ABB RAPID module: Module1.mod

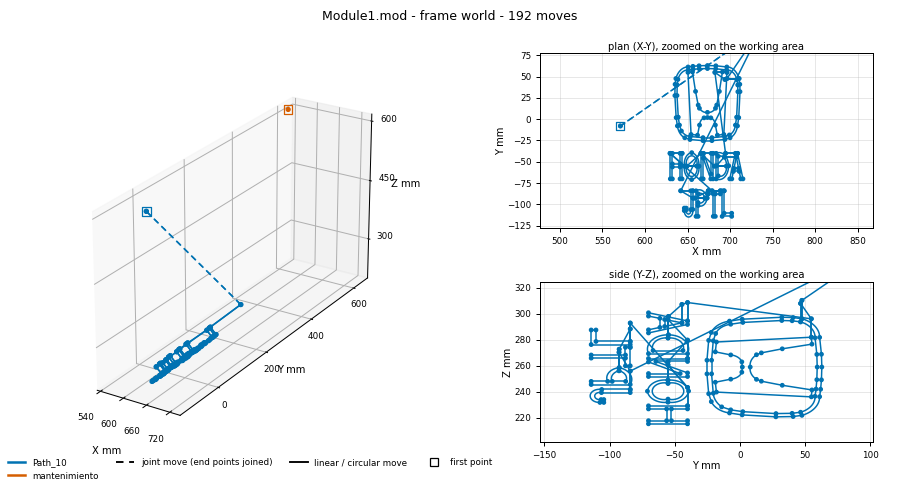
[picture p0: tool path of Module1.mod in frame world, 192 of 192 moves have a stored position in this frame; points joined in program order, loops and branches not executed]
MODULE Module1
        CONST robtarget Target_10:=[[0,0,-20],[0.707106781,0,0,0.707106781],[0,0,0,0],[9E+09,9E+09,9E+09,9E+09,9E+09,9E+09]];
    CONST robtarget Target_20:=[[59.453,57.54,-20],[0.707106781,0,0,0.707106781],[0,0,0,0],[9E+09,9E+09,9E+09,9E+09,9E+09,9E+09]];
    CONST robtarget Target_30:=[[59.453,57.54,0],[0.707106781,0,0,0.707106781],[0,0,0,0],[9E+09,9E+09,9E+09,9E+09,9E+09,9E+09]];
    CONST robtarget Target_40:=[[66.223,56.236,0],[0.707106781,0,0,0.707106781],[0,0,0,0],[9E+09,9E+09,9E+09,9E+09,9E+09,9E+09]];
    CONST robtarget Target_50:=[[74.887,55.915,0],[0.707106781,0,0,0.707106781],[0,0,0,0],[9E+09,9E+09,9E+09,9E+09,9E+09,9E+09]];
    CONST robtarget Target_60:=[[105.351,58.027,0],[0.707106781,0,0,0.707106781],[0,0,0,0],[9E+09,9E+09,9E+09,9E+09,9E+09,9E+09]];
    CONST robtarget Target_70:=[[115.083,60.098,0],[0.707106781,0,0,0.707106781],[0,0,0,0],[9E+09,9E+09,9E+09,9E+09,9E+09,9E+09]];
    CONST robtarget Target_90:=[[123.324,63.988,0],[0.707106781,0,0,0.707106781],[0,0,0,0],[9E+09,9E+09,9E+09,9E+09,9E+09,9E+09]];
    CONST robtarget Target_100:=[[129.054,72.401,0],[0.707106781,0,0,0.707106781],[0,0,0,0],[9E+09,9E+09,9E+09,9E+09,9E+09,9E+09]];
    CONST robtarget Target_110:=[[131.081,81.035,0],[0.707106781,0,0,0.707106781],[0,0,0,0],[9E+09,9E+09,9E+09,9E+09,9E+09,9E+09]];
    CONST robtarget Target_120:=[[132.397,102.578,0],[0.707106781,0,0,0.707106781],[0,0,0,0],[9E+09,9E+09,9E+09,9E+09,9E+09,9E+09]];
    CONST robtarget Target_130:=[[132.397,117.423,0],[0.707106781,0,0,0.707106781],[0,0,0,0],[9E+09,9E+09,9E+09,9E+09,9E+09,9E+09]];
    CONST robtarget Target_140:=[[131.081,138.966,0],[0.707106781,0,0,0.707106781],[0,0,0,0],[9E+09,9E+09,9E+09,9E+09,9E+09,9E+09]];
    CONST robtarget Target_150:=[[129.054,147.6,0],[0.707106781,0,0,0.707106781],[0,0,0,0],[9E+09,9E+09,9E+09,9E+09,9E+09,9E+09]];
    CONST robtarget Target_160:=[[123.324,156.012,0],[0.707106781,0,0,0.707106781],[0,0,0,0],[9E+09,9E+09,9E+09,9E+09,9E+09,9E+09]];
    CONST robtarget Target_170:=[[115.083,159.903,0],[0.707106781,0,0,0.707106781],[0,0,0,0],[9E+09,9E+09,9E+09,9E+09,9E+09,9E+09]];
    CONST robtarget Target_180:=[[105.351,161.974,0],[0.707106781,0,0,0.707106781],[0,0,0,0],[9E+09,9E+09,9E+09,9E+09,9E+09,9E+09]];
    CONST robtarget Target_190:=[[79.466,164.086,0],[0.707106781,0,0,0.707106781],[0,0,0,0],[9E+09,9E+09,9E+09,9E+09,9E+09,9E+09]];
    CONST robtarget Target_200:=[[66.223,163.764,0],[0.707106781,0,0,0.707106781],[0,0,0,0],[9E+09,9E+09,9E+09,9E+09,9E+09,9E+09]];
    CONST robtarget Target_210:=[[59.453,162.461,0],[0.707106781,0,0,0.707106781],[0,0,0,0],[9E+09,9E+09,9E+09,9E+09,9E+09,9E+09]];
    CONST robtarget Target_220:=[[48.886,153.475,0],[0.707106781,0,0,0.707106781],[0,0,0,0],[9E+09,9E+09,9E+09,9E+09,9E+09,9E+09]];
    CONST robtarget Target_230:=[[45.864,142.196,0],[0.707106781,0,0,0.707106781],[0,0,0,0],[9E+09,9E+09,9E+09,9E+09,9E+09,9E+09]];
    CONST robtarget Target_240:=[[45.105,134.144,0],[0.707106781,0,0,0.707106781],[0,0,0,0],[9E+09,9E+09,9E+09,9E+09,9E+09,9E+09]];
    CONST robtarget Target_250:=[[44.474,123.905,0],[0.707106781,0,0,0.707106781],[0,0,0,0],[9E+09,9E+09,9E+09,9E+09,9E+09,9E+09]];
    CONST robtarget Target_260:=[[44.178,110,0],[0.707106781,0,0,0.707106781],[0,0,0,0],[9E+09,9E+09,9E+09,9E+09,9E+09,9E+09]];
    CONST robtarget Target_270:=[[44.474,96.095,0],[0.707106781,0,0,0.707106781],[0,0,0,0],[9E+09,9E+09,9E+09,9E+09,9E+09,9E+09]];
    CONST robtarget Target_280:=[[45.864,77.804,0],[0.707106781,0,0,0.707106781],[0,0,0,0],[9E+09,9E+09,9E+09,9E+09,9E+09,9E+09]];
    CONST robtarget Target_290:=[[48.886,66.526,0],[0.707106781,0,0,0.707106781],[0,0,0,0],[9E+09,9E+09,9E+09,9E+09,9E+09,9E+09]];
    CONST robtarget Target_300:=[[59.453,57.54,0],[0.707106781,0,0,0.707106781],[0,0,0,0],[9E+09,9E+09,9E+09,9E+09,9E+09,9E+09]];
    CONST robtarget Target_310:=[[59.453,57.54,-20],[0.707106781,0,0,0.707106781],[0,0,0,0],[9E+09,9E+09,9E+09,9E+09,9E+09,9E+09]];
    CONST robtarget Target_320:=[[60.499,60.925,-20],[0.707106781,0,0,0.707106781],[0,0,0,0],[9E+09,9E+09,9E+09,9E+09,9E+09,9E+09]];
    CONST robtarget Target_330:=[[60.499,60.925,0],[0.707106781,0,0,0.707106781],[0,0,0,0],[9E+09,9E+09,9E+09,9E+09,9E+09,9E+09]];
    CONST robtarget Target_340:=[[67.002,59.732,0],[0.707106781,0,0,0.707106781],[0,0,0,0],[9E+09,9E+09,9E+09,9E+09,9E+09,9E+09]];
    CONST robtarget Target_350:=[[74.944,59.458,0],[0.707106781,0,0,0.707106781],[0,0,0,0],[9E+09,9E+09,9E+09,9E+09,9E+09,9E+09]];
    CONST robtarget Target_360:=[[104.86,61.536,0],[0.707106781,0,0,0.707106781],[0,0,0,0],[9E+09,9E+09,9E+09,9E+09,9E+09,9E+09]];
    CONST robtarget Target_370:=[[114.154,63.519,0],[0.707106781,0,0,0.707106781],[0,0,0,0],[9E+09,9E+09,9E+09,9E+09,9E+09,9E+09]];
    CONST robtarget Target_380:=[[121.091,66.742,0],[0.707106781,0,0,0.707106781],[0,0,0,0],[9E+09,9E+09,9E+09,9E+09,9E+09,9E+09]];
    CONST robtarget Target_390:=[[125.713,73.58,0],[0.707106781,0,0,0.707106781],[0,0,0,0],[9E+09,9E+09,9E+09,9E+09,9E+09,9E+09]];
    CONST robtarget Target_400:=[[127.565,81.47,0],[0.707106781,0,0,0.707106781],[0,0,0,0],[9E+09,9E+09,9E+09,9E+09,9E+09,9E+09]];
    CONST robtarget Target_410:=[[128.854,102.618,0],[0.707106781,0,0,0.707106781],[0,0,0,0],[9E+09,9E+09,9E+09,9E+09,9E+09,9E+09]];
    CONST robtarget Target_420:=[[128.854,117.382,0],[0.707106781,0,0,0.707106781],[0,0,0,0],[9E+09,9E+09,9E+09,9E+09,9E+09,9E+09]];
    CONST robtarget Target_430:=[[127.565,138.53,0],[0.707106781,0,0,0.707106781],[0,0,0,0],[9E+09,9E+09,9E+09,9E+09,9E+09,9E+09]];
    CONST robtarget Target_440:=[[125.713,146.42,0],[0.707106781,0,0,0.707106781],[0,0,0,0],[9E+09,9E+09,9E+09,9E+09,9E+09,9E+09]];
    CONST robtarget Target_450:=[[121.091,153.258,0],[0.707106781,0,0,0.707106781],[0,0,0,0],[9E+09,9E+09,9E+09,9E+09,9E+09,9E+09]];
    CONST robtarget Target_460:=[[114.154,156.482,0],[0.707106781,0,0,0.707106781],[0,0,0,0],[9E+09,9E+09,9E+09,9E+09,9E+09,9E+09]];
    CONST robtarget Target_470:=[[104.86,158.465,0],[0.707106781,0,0,0.707106781],[0,0,0,0],[9E+09,9E+09,9E+09,9E+09,9E+09,9E+09]];
    CONST robtarget Target_480:=[[79.395,160.544,0],[0.707106781,0,0,0.707106781],[0,0,0,0],[9E+09,9E+09,9E+09,9E+09,9E+09,9E+09]];
    CONST robtarget Target_490:=[[67.002,160.268,0],[0.707106781,0,0,0.707106781],[0,0,0,0],[9E+09,9E+09,9E+09,9E+09,9E+09,9E+09]];
    CONST robtarget Target_500:=[[60.499,159.075,0],[0.707106781,0,0,0.707106781],[0,0,0,0],[9E+09,9E+09,9E+09,9E+09,9E+09,9E+09]];
    CONST robtarget Target_510:=[[52.059,151.898,0],[0.707106781,0,0,0.707106781],[0,0,0,0],[9E+09,9E+09,9E+09,9E+09,9E+09,9E+09]];
    CONST robtarget Target_520:=[[49.379,141.75,0],[0.707106781,0,0,0.707106781],[0,0,0,0],[9E+09,9E+09,9E+09,9E+09,9E+09,9E+09]];
    CONST robtarget Target_530:=[[48.642,133.935,0],[0.707106781,0,0,0.707106781],[0,0,0,0],[9E+09,9E+09,9E+09,9E+09,9E+09,9E+09]];
    CONST robtarget Target_540:=[[48.013,123.721,0],[0.707106781,0,0,0.707106781],[0,0,0,0],[9E+09,9E+09,9E+09,9E+09,9E+09,9E+09]];
    CONST robtarget Target_550:=[[47.721,110,0],[0.707106781,0,0,0.707106781],[0,0,0,0],[9E+09,9E+09,9E+09,9E+09,9E+09,9E+09]];
    CONST robtarget Target_560:=[[48.013,96.28,0],[0.707106781,0,0,0.707106781],[0,0,0,0],[9E+09,9E+09,9E+09,9E+09,9E+09,9E+09]];
    CONST robtarget Target_570:=[[49.379,78.251,0],[0.707106781,0,0,0.707106781],[0,0,0,0],[9E+09,9E+09,9E+09,9E+09,9E+09,9E+09]];
    CONST robtarget Target_580:=[[52.059,68.102,0],[0.707106781,0,0,0.707106781],[0,0,0,0],[9E+09,9E+09,9E+09,9E+09,9E+09,9E+09]];
    CONST robtarget Target_590:=[[60.499,60.925,0],[0.707106781,0,0,0.707106781],[0,0,0,0],[9E+09,9E+09,9E+09,9E+09,9E+09,9E+09]];
    CONST robtarget Target_600:=[[60.499,60.925,-20],[0.707106781,0,0,0.707106781],[0,0,0,0],[9E+09,9E+09,9E+09,9E+09,9E+09,9E+09]];
    CONST robtarget Target_610:=[[52.233,77.609,-20],[0.707106781,0,0,0.707106781],[0,0,0,0],[9E+09,9E+09,9E+09,9E+09,9E+09,9E+09]];
    CONST robtarget Target_620:=[[52.233,77.609,0],[0.707106781,0,0,0.707106781],[0,0,0,0],[9E+09,9E+09,9E+09,9E+09,9E+09,9E+09]];
    CONST robtarget Target_630:=[[125.12,82.794,0],[0.707106781,0,0,0.707106781],[0,0,0,0],[9E+09,9E+09,9E+09,9E+09,9E+09,9E+09]];
    CONST robtarget Target_640:=[[125.974,93.513,0],[0.707106781,0,0,0.707106781],[0,0,0,0],[9E+09,9E+09,9E+09,9E+09,9E+09,9E+09]];
    CONST robtarget Target_650:=[[114.117,96.833,0],[0.707106781,0,0,0.707106781],[0,0,0,0],[9E+09,9E+09,9E+09,9E+09,9E+09,9E+09]];
    CONST robtarget Target_660:=[[109.268,98.854,0],[0.707106781,0,0,0.707106781],[0,0,0,0],[9E+09,9E+09,9E+09,9E+09,9E+09,9E+09]];
    CONST robtarget Target_670:=[[105.623,104.378,0],[0.707106781,0,0,0.707106781],[0,0,0,0],[9E+09,9E+09,9E+09,9E+09,9E+09,9E+09]];
    CONST robtarget Target_680:=[[105.23,110,0],[0.707106781,0,0,0.707106781],[0,0,0,0],[9E+09,9E+09,9E+09,9E+09,9E+09,9E+09]];
    CONST robtarget Target_690:=[[105.623,115.622,0],[0.707106781,0,0,0.707106781],[0,0,0,0],[9E+09,9E+09,9E+09,9E+09,9E+09,9E+09]];
    CONST robtarget Target_700:=[[109.268,121.147,0],[0.707106781,0,0,0.707106781],[0,0,0,0],[9E+09,9E+09,9E+09,9E+09,9E+09,9E+09]];
    CONST robtarget Target_710:=[[114.117,123.168,0],[0.707106781,0,0,0.707106781],[0,0,0,0],[9E+09,9E+09,9E+09,9E+09,9E+09,9E+09]];
    CONST robtarget Target_720:=[[125.974,126.488,0],[0.707106781,0,0,0.707106781],[0,0,0,0],[9E+09,9E+09,9E+09,9E+09,9E+09,9E+09]];
    CONST robtarget Target_730:=[[125.12,137.207,0],[0.707106781,0,0,0.707106781],[0,0,0,0],[9E+09,9E+09,9E+09,9E+09,9E+09,9E+09]];
    CONST robtarget Target_740:=[[52.233,142.391,0],[0.707106781,0,0,0.707106781],[0,0,0,0],[9E+09,9E+09,9E+09,9E+09,9E+09,9E+09]];
    CONST robtarget Target_750:=[[51.773,134.866,0],[0.707106781,0,0,0.707106781],[0,0,0,0],[9E+09,9E+09,9E+09,9E+09,9E+09,9E+09]];
    CONST robtarget Target_760:=[[74.57,129.805,0],[0.707106781,0,0,0.707106781],[0,0,0,0],[9E+09,9E+09,9E+09,9E+09,9E+09,9E+09]];
    CONST robtarget Target_770:=[[90.628,125.39,0],[0.707106781,0,0,0.707106781],[0,0,0,0],[9E+09,9E+09,9E+09,9E+09,9E+09,9E+09]];
    CONST robtarget Target_780:=[[94.375,123.358,0],[0.707106781,0,0,0.707106781],[0,0,0,0],[9E+09,9E+09,9E+09,9E+09,9E+09,9E+09]];
    CONST robtarget Target_790:=[[98.757,116.086,0],[0.707106781,0,0,0.707106781],[0,0,0,0],[9E+09,9E+09,9E+09,9E+09,9E+09,9E+09]];
    CONST robtarget Target_800:=[[99.17,110,0],[0.707106781,0,0,0.707106781],[0,0,0,0],[9E+09,9E+09,9E+09,9E+09,9E+09,9E+09]];
    CONST robtarget Target_810:=[[98.757,103.915,0],[0.707106781,0,0,0.707106781],[0,0,0,0],[9E+09,9E+09,9E+09,9E+09,9E+09,9E+09]];
    CONST robtarget Target_820:=[[94.375,96.643,0],[0.707106781,0,0,0.707106781],[0,0,0,0],[9E+09,9E+09,9E+09,9E+09,9E+09,9E+09]];
    CONST robtarget Target_830:=[[90.628,94.611,0],[0.707106781,0,0,0.707106781],[0,0,0,0],[9E+09,9E+09,9E+09,9E+09,9E+09,9E+09]];
    CONST robtarget Target_840:=[[74.57,90.195,0],[0.707106781,0,0,0.707106781],[0,0,0,0],[9E+09,9E+09,9E+09,9E+09,9E+09,9E+09]];
    CONST robtarget Target_850:=[[51.773,85.135,0],[0.707106781,0,0,0.707106781],[0,0,0,0],[9E+09,9E+09,9E+09,9E+09,9E+09,9E+09]];
    CONST robtarget Target_860:=[[52.233,77.609,0],[0.707106781,0,0,0.707106781],[0,0,0,0],[9E+09,9E+09,9E+09,9E+09,9E+09,9E+09]];
    CONST robtarget Target_870:=[[52.233,77.609,-20],[0.707106781,0,0,0.707106781],[0,0,0,0],[9E+09,9E+09,9E+09,9E+09,9E+09,9E+09]];
    CONST robtarget Target_880:=[[147.311,59.932,-20],[0.707106781,0,0,0.707106781],[0,0,0,0],[9E+09,9E+09,9E+09,9E+09,9E+09,9E+09]];
    CONST robtarget Target_890:=[[147.311,59.932,0],[0.707106781,0,0,0.707106781],[0,0,0,0],[9E+09,9E+09,9E+09,9E+09,9E+09,9E+09]];
    CONST robtarget Target_900:=[[177.311,51.036,0],[0.707106781,0,0,0.707106781],[0,0,0,0],[9E+09,9E+09,9E+09,9E+09,9E+09,9E+09]];
    CONST robtarget Target_910:=[[177.311,54.661,0],[0.707106781,0,0,0.707106781],[0,0,0,0],[9E+09,9E+09,9E+09,9E+09,9E+09,9E+09]];
    CONST robtarget Target_920:=[[168.583,57.094,0],[0.707106781,0,0,0.707106781],[0,0,0,0],[9E+09,9E+09,9E+09,9E+09,9E+09,9E+09]];
    CONST robtarget Target_930:=[[168.583,66.943,0],[0.707106781,0,0,0.707106781],[0,0,0,0],[9E+09,9E+09,9E+09,9E+09,9E+09,9E+09]];
    CONST robtarget Target_940:=[[177.311,69.542,0],[0.707106781,0,0,0.707106781],[0,0,0,0],[9E+09,9E+09,9E+09,9E+09,9E+09,9E+09]];
    CONST robtarget Target_950:=[[177.311,72.976,0],[0.707106781,0,0,0.707106781],[0,0,0,0],[9E+09,9E+09,9E+09,9E+09,9E+09,9E+09]];
    CONST robtarget Target_960:=[[147.311,63.747,0],[0.707106781,0,0,0.707106781],[0,0,0,0],[9E+09,9E+09,9E+09,9E+09,9E+09,9E+09]];
    CONST robtarget Target_970:=[[147.311,59.932,0],[0.707106781,0,0,0.707106781],[0,0,0,0],[9E+09,9E+09,9E+09,9E+09,9E+09,9E+09]];
    CONST robtarget Target_980:=[[147.311,59.932,-20],[0.707106781,0,0,0.707106781],[0,0,0,0],[9E+09,9E+09,9E+09,9E+09,9E+09,9E+09]];
    CONST robtarget Target_990:=[[151.627,61.982,-20],[0.707106781,0,0,0.707106781],[0,0,0,0],[9E+09,9E+09,9E+09,9E+09,9E+09,9E+09]];
    CONST robtarget Target_1000:=[[151.627,61.982,0],[0.707106781,0,0,0.707106781],[0,0,0,0],[9E+09,9E+09,9E+09,9E+09,9E+09,9E+09]];
    CONST robtarget Target_1010:=[[164.91,65.941,0],[0.707106781,0,0,0.707106781],[0,0,0,0],[9E+09,9E+09,9E+09,9E+09,9E+09,9E+09]];
    CONST robtarget Target_1020:=[[164.91,58.31,0],[0.707106781,0,0,0.707106781],[0,0,0,0],[9E+09,9E+09,9E+09,9E+09,9E+09,9E+09]];
    CONST robtarget Target_1030:=[[151.627,61.982,0],[0.707106781,0,0,0.707106781],[0,0,0,0],[9E+09,9E+09,9E+09,9E+09,9E+09,9E+09]];
    CONST robtarget Target_1040:=[[151.627,61.982,-20],[0.707106781,0,0,0.707106781],[0,0,0,0],[9E+09,9E+09,9E+09,9E+09,9E+09,9E+09]];
    CONST robtarget Target_1050:=[[161.977,75.051,-20],[0.707106781,0,0,0.707106781],[0,0,0,0],[9E+09,9E+09,9E+09,9E+09,9E+09,9E+09]];
    CONST robtarget Target_1060:=[[161.977,75.051,0],[0.707106781,0,0,0.707106781],[0,0,0,0],[9E+09,9E+09,9E+09,9E+09,9E+09,9E+09]];
    CONST robtarget Target_1070:=[[177.311,85.567,0],[0.707106781,0,0,0.707106781],[0,0,0,0],[9E+09,9E+09,9E+09,9E+09,9E+09,9E+09]];
    CONST robtarget Target_1080:=[[177.311,95.44,0],[0.707106781,0,0,0.707106781],[0,0,0,0],[9E+09,9E+09,9E+09,9E+09,9E+09,9E+09]];
    CONST robtarget Target_1090:=[[147.311,95.44,0],[0.707106781,0,0,0.707106781],[0,0,0,0],[9E+09,9E+09,9E+09,9E+09,9E+09,9E+09]];
    CONST robtarget Target_1100:=[[147.311,85.424,0],[0.707106781,0,0,0.707106781],[0,0,0,0],[9E+09,9E+09,9E+09,9E+09,9E+09,9E+09]];
    CONST robtarget Target_1110:=[[161.977,75.051,0],[0.707106781,0,0,0.707106781],[0,0,0,0],[9E+09,9E+09,9E+09,9E+09,9E+09,9E+09]];
    CONST robtarget Target_1120:=[[161.977,75.051,-20],[0.707106781,0,0,0.707106781],[0,0,0,0],[9E+09,9E+09,9E+09,9E+09,9E+09,9E+09]];
    CONST robtarget Target_1130:=[[162.311,78.437,-20],[0.707106781,0,0,0.707106781],[0,0,0,0],[9E+09,9E+09,9E+09,9E+09,9E+09,9E+09]];
    CONST robtarget Target_1140:=[[162.311,78.437,0],[0.707106781,0,0,0.707106781],[0,0,0,0],[9E+09,9E+09,9E+09,9E+09,9E+09,9E+09]];
    CONST robtarget Target_1150:=[[173.806,85.591,0],[0.707106781,0,0,0.707106781],[0,0,0,0],[9E+09,9E+09,9E+09,9E+09,9E+09,9E+09]];
    CONST robtarget Target_1160:=[[173.806,92.054,0],[0.707106781,0,0,0.707106781],[0,0,0,0],[9E+09,9E+09,9E+09,9E+09,9E+09,9E+09]];
    CONST robtarget Target_1170:=[[150.817,92.054,0],[0.707106781,0,0,0.707106781],[0,0,0,0],[9E+09,9E+09,9E+09,9E+09,9E+09,9E+09]];
    CONST robtarget Target_1180:=[[150.817,85.806,0],[0.707106781,0,0,0.707106781],[0,0,0,0],[9E+09,9E+09,9E+09,9E+09,9E+09,9E+09]];
    CONST robtarget Target_1190:=[[162.311,78.437,0],[0.707106781,0,0,0.707106781],[0,0,0,0],[9E+09,9E+09,9E+09,9E+09,9E+09,9E+09]];
    CONST robtarget Target_1200:=[[162.311,78.437,-20],[0.707106781,0,0,0.707106781],[0,0,0,0],[9E+09,9E+09,9E+09,9E+09,9E+09,9E+09]];
    CONST robtarget Target_1210:=[[147.311,100.734,-20],[0.707106781,0,0,0.707106781],[0,0,0,0],[9E+09,9E+09,9E+09,9E+09,9E+09,9E+09]];
    CONST robtarget Target_1220:=[[147.311,100.734,0],[0.707106781,0,0,0.707106781],[0,0,0,0],[9E+09,9E+09,9E+09,9E+09,9E+09,9E+09]];
    CONST robtarget Target_1230:=[[177.311,100.734,0],[0.707106781,0,0,0.707106781],[0,0,0,0],[9E+09,9E+09,9E+09,9E+09,9E+09,9E+09]];
    CONST robtarget Target_1240:=[[177.311,104.455,0],[0.707106781,0,0,0.707106781],[0,0,0,0],[9E+09,9E+09,9E+09,9E+09,9E+09,9E+09]];
    CONST robtarget Target_1250:=[[152.963,117.07,0],[0.707106781,0,0,0.707106781],[0,0,0,0],[9E+09,9E+09,9E+09,9E+09,9E+09,9E+09]];
    CONST robtarget Target_1260:=[[177.311,117.07,0],[0.707106781,0,0,0.707106781],[0,0,0,0],[9E+09,9E+09,9E+09,9E+09,9E+09,9E+09]];
    CONST robtarget Target_1270:=[[177.311,120.289,0],[0.707106781,0,0,0.707106781],[0,0,0,0],[9E+09,9E+09,9E+09,9E+09,9E+09,9E+09]];
    CONST robtarget Target_1280:=[[147.311,120.289,0],[0.707106781,0,0,0.707106781],[0,0,0,0],[9E+09,9E+09,9E+09,9E+09,9E+09,9E+09]];
    CONST robtarget Target_1290:=[[147.311,116.354,0],[0.707106781,0,0,0.707106781],[0,0,0,0],[9E+09,9E+09,9E+09,9E+09,9E+09,9E+09]];
    CONST robtarget Target_1300:=[[171.659,103.954,0],[0.707106781,0,0,0.707106781],[0,0,0,0],[9E+09,9E+09,9E+09,9E+09,9E+09,9E+09]];
    CONST robtarget Target_1310:=[[147.311,103.954,0],[0.707106781,0,0,0.707106781],[0,0,0,0],[9E+09,9E+09,9E+09,9E+09,9E+09,9E+09]];
    CONST robtarget Target_1320:=[[147.311,100.734,0],[0.707106781,0,0,0.707106781],[0,0,0,0],[9E+09,9E+09,9E+09,9E+09,9E+09,9E+09]];
    CONST robtarget Target_1330:=[[147.311,100.734,-20],[0.707106781,0,0,0.707106781],[0,0,0,0],[9E+09,9E+09,9E+09,9E+09,9E+09,9E+09]];
    CONST robtarget Target_1340:=[[162.359,124.272,-20],[0.707106781,0,0,0.707106781],[0,0,0,0],[9E+09,9E+09,9E+09,9E+09,9E+09,9E+09]];
    CONST robtarget Target_1350:=[[162.359,124.272,0],[0.707106781,0,0,0.707106781],[0,0,0,0],[9E+09,9E+09,9E+09,9E+09,9E+09,9E+09]];
    CONST robtarget Target_1360:=[[174.306,127.992,0],[0.707106781,0,0,0.707106781],[0,0,0,0],[9E+09,9E+09,9E+09,9E+09,9E+09,9E+09]];
    CONST robtarget Target_1370:=[[178.098,136.243,0],[0.707106781,0,0,0.707106781],[0,0,0,0],[9E+09,9E+09,9E+09,9E+09,9E+09,9E+09]];
    CONST robtarget Target_1380:=[[174.306,144.494,0],[0.707106781,0,0,0.707106781],[0,0,0,0],[9E+09,9E+09,9E+09,9E+09,9E+09,9E+09]];
    CONST robtarget Target_1390:=[[162.359,148.215,0],[0.707106781,0,0,0.707106781],[0,0,0,0],[9E+09,9E+09,9E+09,9E+09,9E+09,9E+09]];
    CONST robtarget Target_1400:=[[150.316,144.494,0],[0.707106781,0,0,0.707106781],[0,0,0,0],[9E+09,9E+09,9E+09,9E+09,9E+09,9E+09]];
    CONST robtarget Target_1410:=[[146.524,136.076,0],[0.707106781,0,0,0.707106781],[0,0,0,0],[9E+09,9E+09,9E+09,9E+09,9E+09,9E+09]];
    CONST robtarget Target_1420:=[[153.416,126.06,0],[0.707106781,0,0,0.707106781],[0,0,0,0],[9E+09,9E+09,9E+09,9E+09,9E+09,9E+09]];
    CONST robtarget Target_1430:=[[162.359,124.272,0],[0.707106781,0,0,0.707106781],[0,0,0,0],[9E+09,9E+09,9E+09,9E+09,9E+09,9E+09]];
    CONST robtarget Target_1440:=[[162.359,124.272,-20],[0.707106781,0,0,0.707106781],[0,0,0,0],[9E+09,9E+09,9E+09,9E+09,9E+09,9E+09]];
    CONST robtarget Target_1450:=[[162.311,127.658,-20],[0.707106781,0,0,0.707106781],[0,0,0,0],[9E+09,9E+09,9E+09,9E+09,9E+09,9E+09]];
    CONST robtarget Target_1460:=[[162.311,127.658,0],[0.707106781,0,0,0.707106781],[0,0,0,0],[9E+09,9E+09,9E+09,9E+09,9E+09,9E+09]];
    CONST robtarget Target_1470:=[[174.426,136.243,0],[0.707106781,0,0,0.707106781],[0,0,0,0],[9E+09,9E+09,9E+09,9E+09,9E+09,9E+09]];
    CONST robtarget Target_1480:=[[162.311,144.828,0],[0.707106781,0,0,0.707106781],[0,0,0,0],[9E+09,9E+09,9E+09,9E+09,9E+09,9E+09]];
    CONST robtarget Target_1490:=[[150.197,136.339,0],[0.707106781,0,0,0.707106781],[0,0,0,0],[9E+09,9E+09,9E+09,9E+09,9E+09,9E+09]];
    CONST robtarget Target_1500:=[[162.311,127.658,0],[0.707106781,0,0,0.707106781],[0,0,0,0],[9E+09,9E+09,9E+09,9E+09,9E+09,9E+09]];
    CONST robtarget Target_1510:=[[162.311,127.658,-20],[0.707106781,0,0,0.707106781],[0,0,0,0],[9E+09,9E+09,9E+09,9E+09,9E+09,9E+09]];
    CONST robtarget Target_1520:=[[147.311,152.102,-20],[0.707106781,0,0,0.707106781],[0,0,0,0],[9E+09,9E+09,9E+09,9E+09,9E+09,9E+09]];
    CONST robtarget Target_1530:=[[147.311,152.102,0],[0.707106781,0,0,0.707106781],[0,0,0,0],[9E+09,9E+09,9E+09,9E+09,9E+09,9E+09]];
    CONST robtarget Target_1540:=[[177.311,152.102,0],[0.707106781,0,0,0.707106781],[0,0,0,0],[9E+09,9E+09,9E+09,9E+09,9E+09,9E+09]];
    CONST robtarget Target_1550:=[[177.311,155.488,0],[0.707106781,0,0,0.707106781],[0,0,0,0],[9E+09,9E+09,9E+09,9E+09,9E+09,9E+09]];
    CONST robtarget Target_1560:=[[163.36,155.488,0],[0.707106781,0,0,0.707106781],[0,0,0,0],[9E+09,9E+09,9E+09,9E+09,9E+09,9E+09]];
    CONST robtarget Target_1570:=[[163.36,168.27,0],[0.707106781,0,0,0.707106781],[0,0,0,0],[9E+09,9E+09,9E+09,9E+09,9E+09,9E+09]];
    CONST robtarget Target_1580:=[[177.311,168.27,0],[0.707106781,0,0,0.707106781],[0,0,0,0],[9E+09,9E+09,9E+09,9E+09,9E+09,9E+09]];
    CONST robtarget Target_1590:=[[177.311,171.656,0],[0.707106781,0,0,0.707106781],[0,0,0,0],[9E+09,9E+09,9E+09,9E+09,9E+09,9E+09]];
    CONST robtarget Target_1600:=[[147.311,171.656,0],[0.707106781,0,0,0.707106781],[0,0,0,0],[9E+09,9E+09,9E+09,9E+09,9E+09,9E+09]];
    CONST robtarget Target_1610:=[[147.311,168.27,0],[0.707106781,0,0,0.707106781],[0,0,0,0],[9E+09,9E+09,9E+09,9E+09,9E+09,9E+09]];
    CONST robtarget Target_1620:=[[159.688,168.27,0],[0.707106781,0,0,0.707106781],[0,0,0,0],[9E+09,9E+09,9E+09,9E+09,9E+09,9E+09]];
    CONST robtarget Target_1630:=[[159.688,155.488,0],[0.707106781,0,0,0.707106781],[0,0,0,0],[9E+09,9E+09,9E+09,9E+09,9E+09,9E+09]];
    CONST robtarget Target_1640:=[[147.311,155.488,0],[0.707106781,0,0,0.707106781],[0,0,0,0],[9E+09,9E+09,9E+09,9E+09,9E+09,9E+09]];
    CONST robtarget Target_1650:=[[147.311,152.102,0],[0.707106781,0,0,0.707106781],[0,0,0,0],[9E+09,9E+09,9E+09,9E+09,9E+09,9E+09]];
    CONST robtarget Target_1660:=[[147.311,152.102,-20],[0.707106781,0,0,0.707106781],[0,0,0,0],[9E+09,9E+09,9E+09,9E+09,9E+09,9E+09]];
    CONST robtarget Target_1670:=[[191.325,82.201,-20],[0.707106781,0,0,0.707106781],[0,0,0,0],[9E+09,9E+09,9E+09,9E+09,9E+09,9E+09]];
    CONST robtarget Target_1680:=[[191.325,82.201,0],[0.707106781,0,0,0.707106781],[0,0,0,0],[9E+09,9E+09,9E+09,9E+09,9E+09,9E+09]];
    CONST robtarget Target_1690:=[[217.653,82.201,0],[0.707106781,0,0,0.707106781],[0,0,0,0],[9E+09,9E+09,9E+09,9E+09,9E+09,9E+09]];
    CONST robtarget Target_1700:=[[217.653,69.752,0],[0.707106781,0,0,0.707106781],[0,0,0,0],[9E+09,9E+09,9E+09,9E+09,9E+09,9E+09]];
    CONST robtarget Target_1710:=[[221.325,69.752,0],[0.707106781,0,0,0.707106781],[0,0,0,0],[9E+09,9E+09,9E+09,9E+09,9E+09,9E+09]];
    CONST robtarget Target_1720:=[[221.325,85.587,0],[0.707106781,0,0,0.707106781],[0,0,0,0],[9E+09,9E+09,9E+09,9E+09,9E+09,9E+09]];
    CONST robtarget Target_1730:=[[191.325,85.587,0],[0.707106781,0,0,0.707106781],[0,0,0,0],[9E+09,9E+09,9E+09,9E+09,9E+09,9E+09]];
    CONST robtarget Target_1740:=[[191.325,82.201,0],[0.707106781,0,0,0.707106781],[0,0,0,0],[9E+09,9E+09,9E+09,9E+09,9E+09,9E+09]];
    CONST robtarget Target_1750:=[[191.325,82.201,-20],[0.707106781,0,0,0.707106781],[0,0,0,0],[9E+09,9E+09,9E+09,9E+09,9E+09,9E+09]];
    CONST robtarget Target_1760:=[[191.325,88.592,-20],[0.707106781,0,0,0.707106781],[0,0,0,0],[9E+09,9E+09,9E+09,9E+09,9E+09,9E+09]];
    CONST robtarget Target_1770:=[[191.325,88.592,0],[0.707106781,0,0,0.707106781],[0,0,0,0],[9E+09,9E+09,9E+09,9E+09,9E+09,9E+09]];
    CONST robtarget Target_1780:=[[194.998,88.592,0],[0.707106781,0,0,0.707106781],[0,0,0,0],[9E+09,9E+09,9E+09,9E+09,9E+09,9E+09]];
    CONST robtarget Target_1790:=[[194.998,96.915,0],[0.707106781,0,0,0.707106781],[0,0,0,0],[9E+09,9E+09,9E+09,9E+09,9E+09,9E+09]];
    CONST robtarget Target_1800:=[[221.325,96.915,0],[0.707106781,0,0,0.707106781],[0,0,0,0],[9E+09,9E+09,9E+09,9E+09,9E+09,9E+09]];
    CONST robtarget Target_1810:=[[221.325,100.301,0],[0.707106781,0,0,0.707106781],[0,0,0,0],[9E+09,9E+09,9E+09,9E+09,9E+09,9E+09]];
    CONST robtarget Target_1820:=[[194.998,100.301,0],[0.707106781,0,0,0.707106781],[0,0,0,0],[9E+09,9E+09,9E+09,9E+09,9E+09,9E+09]];
    CONST robtarget Target_1830:=[[194.998,108.647,0],[0.707106781,0,0,0.707106781],[0,0,0,0],[9E+09,9E+09,9E+09,9E+09,9E+09,9E+09]];
    CONST robtarget Target_1840:=[[191.325,108.647,0],[0.707106781,0,0,0.707106781],[0,0,0,0],[9E+09,9E+09,9E+09,9E+09,9E+09,9E+09]];
    CONST robtarget Target_1850:=[[191.325,88.592,0],[0.707106781,0,0,0.707106781],[0,0,0,0],[9E+09,9E+09,9E+09,9E+09,9E+09,9E+09]];
    CONST robtarget Target_1860:=[[191.325,88.592,-20],[0.707106781,0,0,0.707106781],[0,0,0,0],[9E+09,9E+09,9E+09,9E+09,9E+09,9E+09]];
    CONST robtarget Target_1870:=[[199.815,110.651,-20],[0.707106781,0,0,0.707106781],[0,0,0,0],[9E+09,9E+09,9E+09,9E+09,9E+09,9E+09]];
    CONST robtarget Target_1880:=[[199.815,110.651,0],[0.707106781,0,0,0.707106781],[0,0,0,0],[9E+09,9E+09,9E+09,9E+09,9E+09,9E+09]];
    CONST robtarget Target_1890:=[[208.662,117.924,0],[0.707106781,0,0,0.707106781],[0,0,0,0],[9E+09,9E+09,9E+09,9E+09,9E+09,9E+09]];
    CONST robtarget Target_1900:=[[208.662,125.579,0],[0.707106781,0,0,0.707106781],[0,0,0,0],[9E+09,9E+09,9E+09,9E+09,9E+09,9E+09]];
    CONST robtarget Target_1910:=[[221.325,125.579,0],[0.707106781,0,0,0.707106781],[0,0,0,0],[9E+09,9E+09,9E+09,9E+09,9E+09,9E+09]];
    CONST robtarget Target_1920:=[[221.325,128.965,0],[0.707106781,0,0,0.707106781],[0,0,0,0],[9E+09,9E+09,9E+09,9E+09,9E+09,9E+09]];
    CONST robtarget Target_1930:=[[191.325,128.965,0],[0.707106781,0,0,0.707106781],[0,0,0,0],[9E+09,9E+09,9E+09,9E+09,9E+09,9E+09]];
    CONST robtarget Target_1940:=[[191.325,117.948,0],[0.707106781,0,0,0.707106781],[0,0,0,0],[9E+09,9E+09,9E+09,9E+09,9E+09,9E+09]];
    CONST robtarget Target_1950:=[[199.815,110.651,0],[0.707106781,0,0,0.707106781],[0,0,0,0],[9E+09,9E+09,9E+09,9E+09,9E+09,9E+09]];
    CONST robtarget Target_1960:=[[199.815,110.651,-20],[0.707106781,0,0,0.707106781],[0,0,0,0],[9E+09,9E+09,9E+09,9E+09,9E+09,9E+09]];
    CONST robtarget Target_1970:=[[199.934,114.037,-20],[0.707106781,0,0,0.707106781],[0,0,0,0],[9E+09,9E+09,9E+09,9E+09,9E+09,9E+09]];
    CONST robtarget Target_1980:=[[199.934,114.037,0],[0.707106781,0,0,0.707106781],[0,0,0,0],[9E+09,9E+09,9E+09,9E+09,9E+09,9E+09]];
    CONST robtarget Target_1990:=[[205.157,119.045,0],[0.707106781,0,0,0.707106781],[0,0,0,0],[9E+09,9E+09,9E+09,9E+09,9E+09,9E+09]];
    CONST robtarget Target_2000:=[[205.157,125.579,0],[0.707106781,0,0,0.707106781],[0,0,0,0],[9E+09,9E+09,9E+09,9E+09,9E+09,9E+09]];
    CONST robtarget Target_2010:=[[194.831,125.579,0],[0.707106781,0,0,0.707106781],[0,0,0,0],[9E+09,9E+09,9E+09,9E+09,9E+09,9E+09]];
    CONST robtarget Target_2020:=[[194.831,118.902,0],[0.707106781,0,0,0.707106781],[0,0,0,0],[9E+09,9E+09,9E+09,9E+09,9E+09,9E+09]];
    CONST robtarget Target_2030:=[[199.934,114.037,0],[0.707106781,0,0,0.707106781],[0,0,0,0],[9E+09,9E+09,9E+09,9E+09,9E+09,9E+09]];
    CONST robtarget Target_2040:=[[199.934,114.037,-20],[0.707106781,0,0,0.707106781],[0,0,0,0],[9E+09,9E+09,9E+09,9E+09,9E+09,9E+09]];
    CONST robtarget Target_2050:=[[191.325,134.379,-20],[0.707106781,0,0,0.707106781],[0,0,0,0],[9E+09,9E+09,9E+09,9E+09,9E+09,9E+09]];
    CONST robtarget Target_2060:=[[191.325,134.379,0],[0.707106781,0,0,0.707106781],[0,0,0,0],[9E+09,9E+09,9E+09,9E+09,9E+09,9E+09]];
    CONST robtarget Target_2070:=[[213.217,134.379,0],[0.707106781,0,0,0.707106781],[0,0,0,0],[9E+09,9E+09,9E+09,9E+09,9E+09,9E+09]];
    CONST robtarget Target_2080:=[[222.112,141.509,0],[0.707106781,0,0,0.707106781],[0,0,0,0],[9E+09,9E+09,9E+09,9E+09,9E+09,9E+09]];
    CONST robtarget Target_2090:=[[214.6,148.449,0],[0.707106781,0,0,0.707106781],[0,0,0,0],[9E+09,9E+09,9E+09,9E+09,9E+09,9E+09]];
    CONST robtarget Target_2100:=[[211.619,148.449,0],[0.707106781,0,0,0.707106781],[0,0,0,0],[9E+09,9E+09,9E+09,9E+09,9E+09,9E+09]];
    CONST robtarget Target_2110:=[[211.619,145.325,0],[0.707106781,0,0,0.707106781],[0,0,0,0],[9E+09,9E+09,9E+09,9E+09,9E+09,9E+09]];
    CONST robtarget Target_2120:=[[213.718,145.325,0],[0.707106781,0,0,0.707106781],[0,0,0,0],[9E+09,9E+09,9E+09,9E+09,9E+09,9E+09]];
    CONST robtarget Target_2130:=[[218.607,141.581,0],[0.707106781,0,0,0.707106781],[0,0,0,0],[9E+09,9E+09,9E+09,9E+09,9E+09,9E+09]];
    CONST robtarget Target_2140:=[[213.432,137.765,0],[0.707106781,0,0,0.707106781],[0,0,0,0],[9E+09,9E+09,9E+09,9E+09,9E+09,9E+09]];
    CONST robtarget Target_2150:=[[191.325,137.765,0],[0.707106781,0,0,0.707106781],[0,0,0,0],[9E+09,9E+09,9E+09,9E+09,9E+09,9E+09]];
    CONST robtarget Target_2160:=[[191.325,134.379,0],[0.707106781,0,0,0.707106781],[0,0,0,0],[9E+09,9E+09,9E+09,9E+09,9E+09,9E+09]];
    CONST robtarget Target_2170:=[[191.325,134.379,-20],[0.707106781,0,0,0.707106781],[0,0,0,0],[9E+09,9E+09,9E+09,9E+09,9E+09,9E+09]];
    CONST robtarget Target_2180:=[[0,0,-20],[0.707106781,0,0,0.707106781],[0,0,0,0],[9E+09,9E+09,9E+09,9E+09,9E+09,9E+09]];
    CONST robtarget Target_5:=[[115.18142236,-41.878607286,-296.515538202],[0.653281482,-0.27059805,0.27059805,0.653281482],[-1,0,-1,0],[9E+09,9E+09,9E+09,9E+09,9E+09,9E+09]];
    CONST robtarget Target_2190:=[[-525.953797687,-36.752575709,-334.376282138],[0.509169636,0.78406871,0.280189062,-0.217891326],[0,-2,0,0],[9E+09,9E+09,9E+09,9E+09,9E+09,9E+09]];
        TASK PERS tooldata prueba1:=[TRUE,[[0,0,0],[1,0,0,0]],[-1,[0,0,0],[1,0,0,0],0,0,0]];
!***********************************************************
    !
    ! M?dulo:  Module1
    !
    ! Descripción:
    !   Trayectorias de dibujo y mantenimiento
    !
    ! Autor: juanp
    !
    ! Versión: 1.0
    !
    !***********************************************************


    !***********************************************************
    !
    ! Procedimiento Main
    !
    !   Este es el punto de entrada de su programa
    !
    !***********************************************************
    PROC main()
        SetDO SalDO_1,0;
        SetDO SalDO_2,0;
        WaitDI EntDI_1,1;
        IF EntDI_1 = 1 SetDO SalDO_1,1;
Path_10;
        WaitDI EntDI_2,1;
        IF EntDI_2 = 1 SetDO SalDO_1,0;
SetDO SalDO_2,1;
mantenimiento;
        SetDO SalDO_2,0;

    ENDPROC
    PROC Path_10()
        MoveJ Target_5,v100,fine,ToolLab4\WObj:=Workobject_1;
        MoveJ Target_10,v100,fine,ToolLab4\WObj:=Workobject_1;
        MoveL Target_20,v100,fine,ToolLab4\WObj:=Workobject_1;
        MoveL Target_30,v100,fine,ToolLab4\WObj:=Workobject_1;
        MoveL Target_40,v100,fine,ToolLab4\WObj:=Workobject_1;
        MoveL Target_50,v100,fine,ToolLab4\WObj:=Workobject_1;
        MoveL Target_60,v100,fine,ToolLab4\WObj:=Workobject_1;
        MoveL Target_70,v100,fine,ToolLab4\WObj:=Workobject_1;
        MoveC Target_90,Target_100,v100,fine,ToolLab4\WObj:=Workobject_1;
        MoveL Target_110,v100,fine,ToolLab4\WObj:=Workobject_1;
        MoveL Target_120,v100,fine,ToolLab4\WObj:=Workobject_1;
        MoveL Target_130,v100,fine,ToolLab4\WObj:=Workobject_1;
        MoveL Target_140,v100,fine,ToolLab4\WObj:=Workobject_1;
        MoveL Target_150,v100,fine,ToolLab4\WObj:=Workobject_1;
        MoveC Target_160,Target_170,v100,fine,ToolLab4\WObj:=Workobject_1;
        MoveL Target_180,v100,fine,ToolLab4\WObj:=Workobject_1;
        MoveL Target_190,v100,fine,ToolLab4\WObj:=Workobject_1;
        MoveL Target_200,v100,fine,ToolLab4\WObj:=Workobject_1;
        MoveL Target_210,v100,fine,ToolLab4\WObj:=Workobject_1;
        MoveC Target_220,Target_230,v100,fine,ToolLab4\WObj:=Workobject_1;
        MoveL Target_240,v100,fine,ToolLab4\WObj:=Workobject_1;
        MoveL Target_250,v100,fine,ToolLab4\WObj:=Workobject_1;
        MoveL Target_260,v100,fine,ToolLab4\WObj:=Workobject_1;
        MoveL Target_270,v100,fine,ToolLab4\WObj:=Workobject_1;
        MoveL Target_280,v100,fine,ToolLab4\WObj:=Workobject_1;
        MoveC Target_290,Target_300,v100,fine,ToolLab4\WObj:=Workobject_1;
        MoveL Target_310,v100,fine,ToolLab4\WObj:=Workobject_1;
        MoveL Target_320,v100,fine,ToolLab4\WObj:=Workobject_1;
        MoveL Target_330,v100,fine,ToolLab4\WObj:=Workobject_1;
        MoveL Target_340,v100,fine,ToolLab4\WObj:=Workobject_1;
        MoveL Target_350,v100,fine,ToolLab4\WObj:=Workobject_1;
        MoveL Target_360,v100,fine,ToolLab4\WObj:=Workobject_1;
        MoveL Target_370,v100,fine,ToolLab4\WObj:=Workobject_1;
        MoveC Target_380,Target_390,v100,fine,ToolLab4\WObj:=Workobject_1;
        MoveL Target_400,v100,fine,ToolLab4\WObj:=Workobject_1;
        MoveL Target_410,v100,fine,ToolLab4\WObj:=Workobject_1;
        MoveL Target_420,v100,fine,ToolLab4\WObj:=Workobject_1;
        MoveL Target_430,v100,fine,ToolLab4\WObj:=Workobject_1;
        MoveC Target_440,Target_450,v100,fine,ToolLab4\WObj:=Workobject_1;
        MoveL Target_460,v100,fine,ToolLab4\WObj:=Workobject_1;
        MoveL Target_470,v100,fine,ToolLab4\WObj:=Workobject_1;
        MoveL Target_480,v100,fine,ToolLab4\WObj:=Workobject_1;
        MoveL Target_490,v100,fine,ToolLab4\WObj:=Workobject_1;
        MoveL Target_500,v100,fine,ToolLab4\WObj:=Workobject_1;
        MoveC Target_510,Target_520,v100,fine,ToolLab4\WObj:=Workobject_1;
        MoveL Target_530,v100,fine,ToolLab4\WObj:=Workobject_1;
        MoveL Target_540,v100,fine,ToolLab4\WObj:=Workobject_1;
        MoveL Target_550,v100,fine,ToolLab4\WObj:=Workobject_1;
        MoveL Target_560,v100,fine,ToolLab4\WObj:=Workobject_1;
        MoveL Target_570,v100,fine,ToolLab4\WObj:=Workobject_1;
        MoveC Target_580,Target_590,v100,fine,ToolLab4\WObj:=Workobject_1;
        MoveL Target_600,v100,fine,ToolLab4\WObj:=Workobject_1;
        MoveL Target_610,v100,fine,ToolLab4\WObj:=Workobject_1;
        MoveL Target_620,v100,fine,ToolLab4\WObj:=Workobject_1;
        MoveL Target_630,v100,fine,ToolLab4\WObj:=Workobject_1;
        MoveL Target_640,v100,fine,ToolLab4\WObj:=Workobject_1;
        MoveL Target_650,v100,fine,ToolLab4\WObj:=Workobject_1;
        MoveC Target_660,Target_670,v100,fine,ToolLab4\WObj:=Workobject_1;
        MoveL Target_680,v100,fine,ToolLab4\WObj:=Workobject_1;
        MoveL Target_690,v100,fine,ToolLab4\WObj:=Workobject_1;
        MoveC Target_700,Target_710,v100,fine,ToolLab4\WObj:=Workobject_1;
        MoveL Target_720,v100,fine,ToolLab4\WObj:=Workobject_1;
        MoveL Target_730,v100,fine,ToolLab4\WObj:=Workobject_1;
        MoveL Target_740,v100,fine,ToolLab4\WObj:=Workobject_1;
        MoveL Target_750,v100,fine,ToolLab4\WObj:=Workobject_1;
        MoveL Target_760,v100,fine,ToolLab4\WObj:=Workobject_1;
        MoveL Target_770,v100,fine,ToolLab4\WObj:=Workobject_1;
        MoveL Target_780,v100,fine,ToolLab4\WObj:=Workobject_1;
        MoveC Target_790,Target_800,v100,fine,ToolLab4\WObj:=Workobject_1;
        MoveC Target_810,Target_820,v100,fine,ToolLab4\WObj:=Workobject_1;
        MoveL Target_830,v100,fine,ToolLab4\WObj:=Workobject_1;
        MoveL Target_840,v100,fine,ToolLab4\WObj:=Workobject_1;
        MoveL Target_850,v100,fine,ToolLab4\WObj:=Workobject_1;
        MoveL Target_860,v100,fine,ToolLab4\WObj:=Workobject_1;
        MoveL Target_870,v100,fine,ToolLab4\WObj:=Workobject_1;
        MoveL Target_880,v100,fine,ToolLab4\WObj:=Workobject_1;
        MoveL Target_890,v100,fine,ToolLab4\WObj:=Workobject_1;
        MoveL Target_900,v100,fine,ToolLab4\WObj:=Workobject_1;
        MoveL Target_910,v100,fine,ToolLab4\WObj:=Workobject_1;
        MoveL Target_920,v100,fine,ToolLab4\WObj:=Workobject_1;
        MoveL Target_930,v100,fine,ToolLab4\WObj:=Workobject_1;
        MoveL Target_940,v100,fine,ToolLab4\WObj:=Workobject_1;
        MoveL Target_950,v100,fine,ToolLab4\WObj:=Workobject_1;
        MoveL Target_960,v100,fine,ToolLab4\WObj:=Workobject_1;
        MoveL Target_970,v100,fine,ToolLab4\WObj:=Workobject_1;
        MoveL Target_980,v100,fine,ToolLab4\WObj:=Workobject_1;
        MoveL Target_990,v100,fine,ToolLab4\WObj:=Workobject_1;
        MoveL Target_1000,v100,fine,ToolLab4\WObj:=Workobject_1;
        MoveL Target_1010,v100,fine,ToolLab4\WObj:=Workobject_1;
        MoveL Target_1020,v100,fine,ToolLab4\WObj:=Workobject_1;
        MoveL Target_1030,v100,fine,ToolLab4\WObj:=Workobject_1;
        MoveL Target_1040,v100,fine,ToolLab4\WObj:=Workobject_1;
        MoveL Target_1050,v100,fine,ToolLab4\WObj:=Workobject_1;
        MoveL Target_1060,v100,fine,ToolLab4\WObj:=Workobject_1;
        MoveC Target_1070,Target_1080,v100,fine,ToolLab4\WObj:=Workobject_1;
        MoveL Target_1090,v100,fine,ToolLab4\WObj:=Workobject_1;
        MoveC Target_1100,Target_1110,v100,fine,ToolLab4\WObj:=Workobject_1;
        MoveL Target_1120,v100,fine,ToolLab4\WObj:=Workobject_1;
        MoveL Target_1130,v100,fine,ToolLab4\WObj:=Workobject_1;
        MoveL Target_1140,v100,fine,ToolLab4\WObj:=Workobject_1;
        MoveC Target_1150,Target_1160,v100,fine,ToolLab4\WObj:=Workobject_1;
        MoveL Target_1170,v100,fine,ToolLab4\WObj:=Workobject_1;
        MoveC Target_1180,Target_1190,v100,fine,ToolLab4\WObj:=Workobject_1;
        MoveL Target_1200,v100,fine,ToolLab4\WObj:=Workobject_1;
        MoveL Target_1210,v100,fine,ToolLab4\WObj:=Workobject_1;
        MoveL Target_1220,v100,fine,ToolLab4\WObj:=Workobject_1;
        MoveL Target_1230,v100,fine,ToolLab4\WObj:=Workobject_1;
        MoveL Target_1240,v100,fine,ToolLab4\WObj:=Workobject_1;
        MoveL Target_1250,v100,fine,ToolLab4\WObj:=Workobject_1;
        MoveL Target_1260,v100,fine,ToolLab4\WObj:=Workobject_1;
        MoveL Target_1270,v100,fine,ToolLab4\WObj:=Workobject_1;
        MoveL Target_1280,v100,fine,ToolLab4\WObj:=Workobject_1;
        MoveL Target_1290,v100,fine,ToolLab4\WObj:=Workobject_1;
        MoveL Target_1300,v100,fine,ToolLab4\WObj:=Workobject_1;
        MoveL Target_1310,v100,fine,ToolLab4\WObj:=Workobject_1;
        MoveL Target_1320,v100,fine,ToolLab4\WObj:=Workobject_1;
        MoveL Target_1330,v100,fine,ToolLab4\WObj:=Workobject_1;
        MoveL Target_1340,v100,fine,ToolLab4\WObj:=Workobject_1;
        MoveL Target_1350,v100,fine,ToolLab4\WObj:=Workobject_1;
        MoveC Target_1360,Target_1370,v100,fine,ToolLab4\WObj:=Workobject_1;
        MoveC Target_1380,Target_1390,v100,fine,ToolLab4\WObj:=Workobject_1;
        MoveC Target_1400,Target_1410,v100,fine,ToolLab4\WObj:=Workobject_1;
        MoveC Target_1420,Target_1430,v100,fine,ToolLab4\WObj:=Workobject_1;
        MoveL Target_1440,v100,fine,ToolLab4\WObj:=Workobject_1;
        MoveL Target_1450,v100,fine,ToolLab4\WObj:=Workobject_1;
        MoveL Target_1460,v100,fine,ToolLab4\WObj:=Workobject_1;
        MoveC Target_1470,Target_1480,v100,fine,ToolLab4\WObj:=Workobject_1;
        MoveC Target_1490,Target_1500,v100,fine,ToolLab4\WObj:=Workobject_1;
        MoveL Target_1510,v100,fine,ToolLab4\WObj:=Workobject_1;
        MoveL Target_1520,v100,fine,ToolLab4\WObj:=Workobject_1;
        MoveL Target_1530,v100,fine,ToolLab4\WObj:=Workobject_1;
        MoveL Target_1540,v100,fine,ToolLab4\WObj:=Workobject_1;
        MoveL Target_1550,v100,fine,ToolLab4\WObj:=Workobject_1;
        MoveL Target_1560,v100,fine,ToolLab4\WObj:=Workobject_1;
        MoveL Target_1570,v100,fine,ToolLab4\WObj:=Workobject_1;
        MoveL Target_1580,v100,fine,ToolLab4\WObj:=Workobject_1;
        MoveL Target_1590,v100,fine,ToolLab4\WObj:=Workobject_1;
        MoveL Target_1600,v100,fine,ToolLab4\WObj:=Workobject_1;
        MoveL Target_1610,v100,fine,ToolLab4\WObj:=Workobject_1;
        MoveL Target_1620,v100,fine,ToolLab4\WObj:=Workobject_1;
        MoveL Target_1630,v100,fine,ToolLab4\WObj:=Workobject_1;
        MoveL Target_1640,v100,fine,ToolLab4\WObj:=Workobject_1;
        MoveL Target_1650,v100,fine,ToolLab4\WObj:=Workobject_1;
        MoveL Target_1660,v100,fine,ToolLab4\WObj:=Workobject_1;
        MoveL Target_1670,v100,fine,ToolLab4\WObj:=Workobject_1;
        MoveL Target_1680,v100,fine,ToolLab4\WObj:=Workobject_1;
        MoveL Target_1690,v100,fine,ToolLab4\WObj:=Workobject_1;
        MoveL Target_1700,v100,fine,ToolLab4\WObj:=Workobject_1;
        MoveL Target_1710,v100,fine,ToolLab4\WObj:=Workobject_1;
        MoveL Target_1720,v100,fine,ToolLab4\WObj:=Workobject_1;
        MoveL Target_1730,v100,fine,ToolLab4\WObj:=Workobject_1;
        MoveL Target_1740,v100,fine,ToolLab4\WObj:=Workobject_1;
        MoveL Target_1750,v100,fine,ToolLab4\WObj:=Workobject_1;
        MoveL Target_1760,v100,fine,ToolLab4\WObj:=Workobject_1;
        MoveL Target_1770,v100,fine,ToolLab4\WObj:=Workobject_1;
        MoveL Target_1780,v100,fine,ToolLab4\WObj:=Workobject_1;
        MoveL Target_1790,v100,fine,ToolLab4\WObj:=Workobject_1;
        MoveL Target_1800,v100,fine,ToolLab4\WObj:=Workobject_1;
        MoveL Target_1810,v100,fine,ToolLab4\WObj:=Workobject_1;
        MoveL Target_1820,v100,fine,ToolLab4\WObj:=Workobject_1;
        MoveL Target_1830,v100,fine,ToolLab4\WObj:=Workobject_1;
        MoveL Target_1840,v100,fine,ToolLab4\WObj:=Workobject_1;
        MoveL Target_1850,v100,fine,ToolLab4\WObj:=Workobject_1;
        MoveL Target_1860,v100,fine,ToolLab4\WObj:=Workobject_1;
        MoveL Target_1870,v100,fine,ToolLab4\WObj:=Workobject_1;
        MoveL Target_1880,v100,fine,ToolLab4\WObj:=Workobject_1;
        MoveC Target_1890,Target_1900,v100,fine,ToolLab4\WObj:=Workobject_1;
        MoveL Target_1910,v100,fine,ToolLab4\WObj:=Workobject_1;
        MoveL Target_1920,v100,fine,ToolLab4\WObj:=Workobject_1;
        MoveL Target_1930,v100,fine,ToolLab4\WObj:=Workobject_1;
        MoveC Target_1940,Target_1950,v100,fine,ToolLab4\WObj:=Workobject_1;
        MoveL Target_1960,v100,fine,ToolLab4\WObj:=Workobject_1;
        MoveL Target_1970,v100,fine,ToolLab4\WObj:=Workobject_1;
        MoveL Target_1980,v100,fine,ToolLab4\WObj:=Workobject_1;
        MoveC Target_1990,Target_2000,v100,fine,ToolLab4\WObj:=Workobject_1;
        MoveL Target_2010,v100,fine,ToolLab4\WObj:=Workobject_1;
        MoveC Target_2020,Target_2030,v100,fine,ToolLab4\WObj:=Workobject_1;
        MoveL Target_2040,v100,fine,ToolLab4\WObj:=Workobject_1;
        MoveL Target_2050,v100,fine,ToolLab4\WObj:=Workobject_1;
        MoveL Target_2060,v100,fine,ToolLab4\WObj:=Workobject_1;
        MoveL Target_2070,v100,fine,ToolLab4\WObj:=Workobject_1;
        MoveC Target_2080,Target_2090,v100,fine,ToolLab4\WObj:=Workobject_1;
        MoveL Target_2100,v100,fine,ToolLab4\WObj:=Workobject_1;
        MoveL Target_2110,v100,fine,ToolLab4\WObj:=Workobject_1;
        MoveL Target_2120,v100,fine,ToolLab4\WObj:=Workobject_1;
        MoveC Target_2130,Target_2140,v100,fine,ToolLab4\WObj:=Workobject_1;
        MoveL Target_2150,v100,fine,ToolLab4\WObj:=Workobject_1;
        MoveL Target_2160,v100,fine,ToolLab4\WObj:=Workobject_1;
        MoveL Target_2170,v100,fine,ToolLab4\WObj:=Workobject_1;
        MoveL Target_2180,v100,fine,ToolLab4\WObj:=Workobject_1;
        MoveJ Target_5,v100,fine,ToolLab4\WObj:=Workobject_1;
    ENDPROC
    PROC mantenimiento()
        MoveJ Target_2190,v100,fine,ToolLab4\WObj:=Workobject_1;
    ENDPROC
ENDMODULE
